// TIA Portal V21 export
VAR_GLOBAL   // PLC tag table "K_Zona_Filler"
END_VAR
VAR_GLOBAL CONSTANT   // user constants
   K_Zona_Filler_Main : Int := 0;
END_VAR
